ABB RobotStudio station: robotstudio与PLC.rsstn

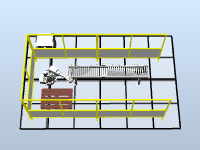
Station Station (saved by RobotStudio 6.8.8148.134)
Controller System2
  mechanical unit ROB_1: IRB2600_12_165_C_01, 6 joints, base frame (0, 0, 0) mm
Layout (positions relative to the parent item):
  - IRB2600_12_165_C_01 [mechanism, from Robots\IRB2600_12_165_C_01.rslib] at (0, 0, 0) mm; joint values [-0.5396, 0.2236, -0.2119, 0.0109, 1.5667, -0.5514] (rad or m)
  - 400_guide [part, from Equipment\Conveyor Guide 400.rslib] at (811.92, -188.84, 0) mm
  - Euro Pallet [graphiccomponentgroup, from Equipment\Euro Pallet.rslib] at (-277.18, -1226.8, 0) mm
    - Body 1 [part, from Equipment\Euro Pallet.rslib]
  - 吸盘夹取 [smart component] at (-618.41, -586.83, 1422.85) mm, rotated rx 1.52 ry 60.04 rz 1.99 deg
      signals: DI xi
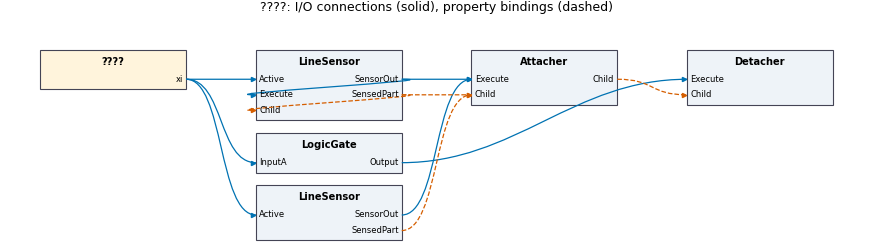
      connections:
        吸盘夹取.xi -> LineSensor.Active
        LineSensor.SensorOut -> Attacher.Execute
        吸盘夹取.xi -> LogicGate.InputA
        LogicGate.Output -> Detacher.Execute
        LineSensor.SensorOut -> Attacher.Execute
        吸盘夹取.xi -> LineSensor.Active
        LineSensor.SensorOut -> Attacher.Execute
        LineSensor.SensedPart => Attacher.Child
        LineSensor.SensedPart => Attacher.Child
        Attacher.Child => Detacher.Child
        LineSensor.SensedPart => Attacher.Child
    - Detacher [smart component, from Components\Detacher.rslib] at (1061.91, 0, 1192.5) mm, rotated rx 180 ry 60 rz 180 deg
        properties: Child=工件示教; KeepPosition=true
    - LogicGate [smart component, from Components\LogicGate.rslib]
        properties: Operator=NOT; Delay=0
    - Attacher [smart component, from Components\Attacher.rslib]
        properties: Parent=MyNewTool; Flange=0; Child=工件示教; Mount=false; Offset=[0 0 0]; Orientation=[0 0 0]
    - MyNewTool [mechanism, from Libraries\吸盘.rslib] at (1018.61, 0, 1217.5) mm, rotated rx 180 ry 60 rz 180 deg
    - LineSensor [smart component, from Components\LineSensor.rslib] at (1061.91, 0, 1192.5) mm, rotated rx 180 ry 60 rz 180 deg
        properties: Start=[-0.0872506979430503 -0.0542341684024924 0.0301000224274997]; End=[-0.0872517349861355 -0.0542607713829768 0.0520446025603243]; Radius=0.008; SensedPart=工件示教; SensedPoint=[-0.051070556640625 -1.17803002929688 0.244311645507813]
      - _sensorPart_ [part]
  - 传送带输送 [smart component]
      signals: DO daowei
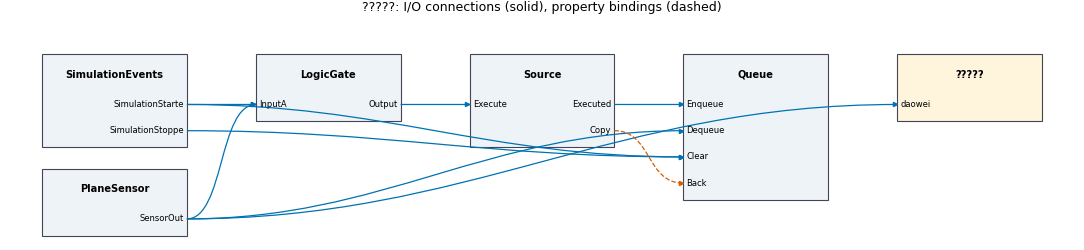
      connections:
        SimulationEvents.SimulationStarted -> LogicGate.InputA
        LogicGate.Output -> Source.Execute
        Source.Executed -> Queue.Enqueue
        PlaneSensor.SensorOut -> Queue.Dequeue
        PlaneSensor.SensorOut -> LogicGate.InputA
        PlaneSensor.SensorOut -> 传送带输送.daowei
        SimulationEvents.SimulationStopped -> Queue.Clear
        SimulationEvents.SimulationStarted -> Queue.Clear
        Source.Copy => Queue.Back
    - Queue [smart component, from Components\Queue.rslib]
        properties: Back=(none); Front=(none); Queue=; NumberOfObjects=0
    - LinearMover [smart component, from Components\LinearMover.rslib]
        properties: Object=Queue; Direction=[-0.001 0 0]; Speed=0.8; Reference=Global; ReferenceObject=(none)
    - PlaneSensor [smart component, from Components\PlaneSensor.rslib]
        properties: Origin=[0.811918 -0.208837 0.77]; Axis1=[0 0.45 0]; Axis2=[0 0 0.08]; SensedPart=(none)
      - _sensorPart_ [part]
    - LogicGate [smart component, from Components\LogicGate.rslib]
        properties: Operator=NOT; Delay=0
    - SimulationEvents [smart component, from Components\SimulationEvents.rslib]
    - Source [smart component, from Components\Source.rslib]
        properties: Source=工件; Copy=(none); Parent=(none); Position=[0 0 0]; Orientation=[0 0 0]; Transient=false; PhysicsBehavior=0
    - 工件 [part] at (1.21, 0, 0) mm
    - 工件示教 [part] at (-2688, 0, 0) mm
  - Fence_2500_4 [graphiccomponentgroup, from Equipment\Fence_2500.rslib] at (4343.47, -1594.28, 3.91) mm, rotated rx 0 ry 0 rz 90 deg
    - Body 1 [part, from Equipment\Fence_2500.rslib]
    - Body 2 [part, from Equipment\Fence_2500.rslib]
  - Fence_2500_5 [graphiccomponentgroup, from Equipment\Fence_2500.rslib] at (-631.95, -1574.22, 0) mm
    - Body 1 [part, from Equipment\Fence_2500.rslib]
    - Body 2 [part, from Equipment\Fence_2500.rslib]
  - Fence_2500_6 [graphiccomponentgroup, from Equipment\Fence_2500.rslib] at (1868.05, -1593.78, 0) mm, rotated rx 0 ry 0 rz 90 deg
    - Body 1 [part, from Equipment\Fence_2500.rslib]
    - Body 2 [part, from Equipment\Fence_2500.rslib]
  - Fence_2500_7 [graphiccomponentgroup, from Equipment\Fence_2500.rslib] at (1868.05, 906.22, 0) mm, rotated rx 0 ry 0 rz 90 deg
    - Body 1 [part, from Equipment\Fence_2500.rslib]
    - Body 2 [part, from Equipment\Fence_2500.rslib]
  - Fence_2500_8 [graphiccomponentgroup, from Equipment\Fence_2500.rslib] at (4368.05, 906.22, 0) mm, rotated rx 0 ry 0 rz 90 deg
    - Body 1 [part, from Equipment\Fence_2500.rslib]
    - Body 2 [part, from Equipment\Fence_2500.rslib]
  - IRC5_Singel-Cabinet [part, from Equipment\IRC5_Singel-Cabinet.rslib] at (-163.45, 1475.26, 82.37) mm, rotated rx 90 ry 0 rz 180 deg
Attachment: Detacher is attached to MyNewTool / 吸盘
Attachment: MyNewTool is attached to IRB2600_12_165_C_01 / Link6
Attachment: LineSensor is attached to MyNewTool / 吸盘
Attachment: 吸盘夹取 is attached to IRB2600_12_165_C_01 / Link6
Station logic (signal -> signal, property => property):
  System2.do1xi -> 吸盘夹取.xi
  传送带输送.daowei -> System2.di1daowei
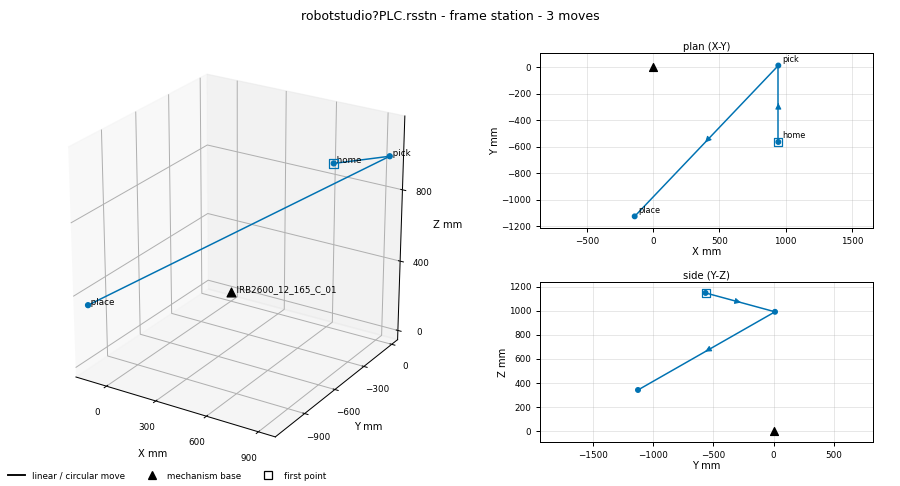
[picture p0: tool path of robotstudio与PLC.rsstn in frame station, 3 of 3 moves have a stored position in this frame; points joined in program order, loops and branches not executed]
Targets, tools, work objects and paths stored in the station, written as RAPID:
! task T_ROB1
MODULE CalibData
  PERS tooldata MyNewTool:=[TRUE,[[0,0,50],[1,0,0,0]],[1,[0,0,1],[1,0,0,0],0,0,0]];
ENDMODULE

! task T_ROB1
MODULE Module1
  CONST robtarget pick:=[[944.920988331,11.894129593,991.590813693],[0.000424818,0.005871422,-0.999960736,-0.006623683],[0,0,-1,0],[9E+09,9E+09,9E+09,9E+09,9E+09,9E+09]];
  CONST robtarget home:=[[944.921000465,-564.843997317,1148.272056966],[0.000424778,0.005871429,-0.999960736,-0.006623676],[-1,0,-1,0],[9E+09,9E+09,9E+09,9E+09,9E+09,9E+09]];
  CONST robtarget place:=[[-138.862555911,-1126.096001158,342.312399035],[0.000424761,0.005871513,-0.999960735,-0.006623749],[-2,-1,-2,0],[9E+09,9E+09,9E+09,9E+09,9E+09,9E+09]];
  PROC Path_10()
    MoveL home,v1000,z100,tool0\WObj:=wobj0;
    MoveL pick,v1000,z100,tool0\WObj:=wobj0;
    MoveL place,v1000,z100,tool0\WObj:=wobj0;
  ENDPROC
ENDMODULE

